(* IEC 61131-3 sources: CodesysTest/export/Unused/FB_SimBasicPrinter.pou, 2 files *)

(* ---- FB_SimBasicPrinter.pou.st ---- *)
(*#-#-#-#-#-#-#-#-#-#---Declaration---#-#-#-#-#-#-#-#-#-#-#-#-#*)

FUNCTION_BLOCK FB_SimBasicPrinter EXTENDS FB_BaseComponent IMPLEMENTS IPrinter, IExecuteAutomatically
VAR_INPUT
	printSpeed : UDINT;
	printLength : REAL;
END_VAR
VAR_OUTPUT
END_VAR
VAR
	beginPrinting : FB_SimulatedFeedback(name := CONCAT(_prefix,'Begin Printing'));
END_VAR
(*#-#-#-#-#-#-#-#-#-#---Implementation---#-#-#-#-#-#-#-#-#-#-#-#-#*)

(* ---- ClearStatus.m.st ---- *)
(*#-#-#-#-#-#-#-#-#-#---Declaration---#-#-#-#-#-#-#-#-#-#-#-#-#*)

METHOD ClearStatus : BOOL
VAR_INPUT
END_VAR
(*#-#-#-#-#-#-#-#-#-#---Implementation---#-#-#-#-#-#-#-#-#-#-#-#-#*)

beginPrinting.in := FALSE;
THIS^.Execute();
